FUNCTION_BLOCK MoveDown EXTENDS GuardMove
VAR_INPUT
END_VAR
VAR_OUTPUT
END_VAR
VAR
END_VAR

(*

short summary
=================
This abstract property returns the class name of the concrete object, 
which is useful for logging/debugging purpose or to check the class name
for ``__DELETE`` in factories (sometimes it's necessary to do more 
than just to free the memory).

.. <legal notes>

legal notes
=================
| SPDX-FileCopyrightText: © 2022 ekvip automation GmbH <info@ekvip.de>
| SPDX-License-Identifier: Apache-2.0
| For details check: Apache-2.0_

.. _Apache-2.0: https://www.apache.org/licenses/LICENSE-2.0

.. </legal notes>

*)
PROPERTY className : CNM_AbstractObject.ClassName
GET
className := 'MoveDown';
END_GET
END_PROPERTY

PROPERTY PROTECTED direction : Rotation
GET
direction := Rotation.DOWN;
END_GET
END_PROPERTY

END_FUNCTION_BLOCK

(* stored: Version 1.1.0.1
   POU MoveDown: Id {eeb5ec9a-c15f-49b0-8576-35711633ef6b}, SpecialFunc None
   Property className: Id {ba179872-1cdf-4400-9795-13710069889a}
   Get Get: Id {79f93b75-720f-4626-b0cc-6422cbb1c694}
   Property direction: Id {1287a1d7-9d31-491e-a7e3-2a7b189b9637}
   Get Get: Id {ed1c390b-7256-4848-9793-800008594aeb} *)
